// TIA Portal V17 export
// export: Created 2025-01-08T13:55:36.0615865Z, ExportSetting WithDefaults, DisplayName Totally Integrated Automation Portal, DisplayVersion V17, DisplayName TIA Portal Openness, DisplayVersion V17, DisplayName TIA Portal Version Control Interface, DisplayVersion V17, DisplayName SINAMICS Startdrive Advanced, DisplayVersion V17 Update2, DisplayName SINAMICS Startdrive G130, G150, S120, S150, SINAMICS MV, S210, DisplayVersion V17 Update2, DisplayName SINAMICS Startdrive G110M, G120, G120C, G120D, G120P, G115D, DisplayVersion V17 Update2, DisplayName STEP 7 Professional, DisplayVersion V17, DisplayName STEP 7 Safety, DisplayVersion V17, DisplayName WinCC Advanced, DisplayVersion V17
TYPE "UDT_Subsystem_Utility"
// stored: IsFailsafeCompliant false
   STRUCT
      Lifebit : Bool;   // Lifebit 1Hz, Check data exchange
      Fault : Bool;   // General Fault
      active : Bool;   // Machine is running or ready
      in_progress : Bool;   // Operation in is progress, motors are running
      EStop : Bool;   // Emergency stop active (1=good)
      General05 : Bool;   // General Signal, Operation mode 05
      General06 : Bool;   // General Signal, Operation mode 06
      General07 : Bool;   // General Signal, Operation mode 07
      General08 : Bool;   // General Signal, Operation mode 08
      General09 : Bool;   // General Signal, Operation mode 09
      General10 : Bool;   // General Signal, Operation mode 10
      General11 : Bool;   // General Signal, Operation mode 11
      General12 : Bool;   // General Signal, Operation mode 12
      General13 : Bool;   // General Signal, Operation mode 13
      General14 : Bool;   // General Signal, Operation mode 14
      General15 : Bool;   // General Signal, Operation mode 15
      Status00 : Bool;   // Motor running, status 00
      Status01 : Bool;   // Motor running, status 01
      Status02 : Bool;   // Motor running, status 02
      Status03 : Bool;   // Motor running, status 03
      Status04 : Bool;   // Motor running, status 04
      Status05 : Bool;   // Motor running, status 05
      Status06 : Bool;   // Motor running, status 06
      Status07 : Bool;   // Motor running, status 07
      Status08 : Bool;   // Motor running, status 08
      Status09 : Bool;   // Motor running, status 09
      Status10 : Bool;   // Motor running, status 10
      Status11 : Bool;   // Motor running, status 11
      Status12 : Bool;   // Motor running, status 12
      Status13 : Bool;   // Motor running, status 13
      Status14 : Bool;   // Motor running, status 14
      Status15 : Bool;   // Motor running, status 15
      Status16 : Bool;   // Motor running, status 16
      Status17 : Bool;   // Motor running, status 17
      Status18 : Bool;   // Motor running, status 18
      Status19 : Bool;   // Motor running, status 19
      Status20 : Bool;   // Motor running, status 20
      Status21 : Bool;   // Motor running, status 21
      Status22 : Bool;   // Motor running, status 22
      Status23 : Bool;   // Motor running, status 23
      Status24 : Bool;   // Motor running, status 24
      Status25 : Bool;   // Motor running, status 25
      Status26 : Bool;   // Motor running, status 26
      Status27 : Bool;   // Motor running, status 27
      Status28 : Bool;   // Motor running, status 28
      Status29 : Bool;   // Motor running, status 29
      Status30 : Bool;   // Motor running, status 30
      Status31 : Bool;   // Motor running, status 31
      Alarm000 : Bool;   // Alarm 0 active
      Alarm001 : Bool;   // Alarm 1 active
      Alarm002 : Bool;   // Alarm 2 active
      Alarm003 : Bool;   // Alarm 3 active
      Alarm004 : Bool;   // Alarm 4 active
      Alarm005 : Bool;   // Alarm 5 active
      Alarm006 : Bool;   // Alarm 6 active
      Alarm007 : Bool;   // Alarm 7 active
      Alarm008 : Bool;   // Alarm 8 active
      Alarm009 : Bool;   // Alarm 9 active
      Alarm010 : Bool;   // Alarm 10 active
      Alarm011 : Bool;   // Alarm 11 active
      Alarm012 : Bool;   // Alarm 12 active
      Alarm013 : Bool;   // Alarm 13 active
      Alarm014 : Bool;   // Alarm 14 active
      Alarm015 : Bool;   // Alarm 15 active
      Alarm016 : Bool;   // Alarm 16 active
      Alarm017 : Bool;   // Alarm 17 active
      Alarm018 : Bool;   // Alarm 18 active
      Alarm019 : Bool;   // Alarm 19 active
      Alarm020 : Bool;   // Alarm 20 active
      Alarm021 : Bool;   // Alarm 21 active
      Alarm022 : Bool;   // Alarm 22 active
      Alarm023 : Bool;   // Alarm 23 active
      Alarm024 : Bool;   // Alarm 24 active
      Alarm025 : Bool;   // Alarm 25 active
      Alarm026 : Bool;   // Alarm 26 active
      Alarm027 : Bool;   // Alarm 27 active
      Alarm028 : Bool;   // Alarm 28 active
      Alarm029 : Bool;   // Alarm 29 active
      Alarm030 : Bool;   // Alarm 30 active
      Alarm031 : Bool;   // Alarm 31 active
      Alarm032 : Bool;   // Alarm 32 active
      Alarm033 : Bool;   // Alarm 33 active
      Alarm034 : Bool;   // Alarm 34 active
      Alarm035 : Bool;   // Alarm 35 active
      Alarm036 : Bool;   // Alarm 36 active
      Alarm037 : Bool;   // Alarm 37 active
      Alarm038 : Bool;   // Alarm 38 active
      Alarm039 : Bool;   // Alarm 39 active
      Alarm040 : Bool;   // Alarm 40 active
      Alarm041 : Bool;   // Alarm 41 active
      Alarm042 : Bool;   // Alarm 42 active
      Alarm043 : Bool;   // Alarm 43 active
      Alarm044 : Bool;   // Alarm 44 active
      Alarm045 : Bool;   // Alarm 45 active
      Alarm046 : Bool;   // Alarm 46 active
      Alarm047 : Bool;   // Alarm 47 active
      Alarm048 : Bool;   // Alarm 48 active
      Alarm049 : Bool;   // Alarm 49 active
      Alarm050 : Bool;   // Alarm 50 active
      Alarm051 : Bool;   // Alarm 51 active
      Alarm052 : Bool;   // Alarm 52 active
      Alarm053 : Bool;   // Alarm 53 active
      Alarm054 : Bool;   // Alarm 54 active
      Alarm055 : Bool;   // Alarm 55 active
      Alarm056 : Bool;   // Alarm 56 active
      Alarm057 : Bool;   // Alarm 57 active
      Alarm058 : Bool;   // Alarm 58 active
      Alarm059 : Bool;   // Alarm 59 active
      Alarm060 : Bool;   // Alarm 60 active
      Alarm061 : Bool;   // Alarm 61 active
      Alarm062 : Bool;   // Alarm 62 active
      Alarm063 : Bool;   // Alarm 63 active
      Alarm064 : Bool;   // Alarm 64 active
      Alarm065 : Bool;   // Alarm 65 active
      Alarm066 : Bool;   // Alarm 66 active
      Alarm067 : Bool;   // Alarm 67 active
      Alarm068 : Bool;   // Alarm 68 active
      Alarm069 : Bool;   // Alarm 69 active
      Alarm070 : Bool;   // Alarm 70 active
      Alarm071 : Bool;   // Alarm 71 active
      Alarm072 : Bool;   // Alarm 72 active
      Alarm073 : Bool;   // Alarm 73 active
      Alarm074 : Bool;   // Alarm 74 active
      Alarm075 : Bool;   // Alarm 75 active
      Alarm076 : Bool;   // Alarm 76 active
      Alarm077 : Bool;   // Alarm 77 active
      Alarm078 : Bool;   // Alarm 78 active
      Alarm079 : Bool;   // Alarm 79 active
      Alarm080 : Bool;   // Alarm 80 active
      Alarm081 : Bool;   // Alarm 81 active
      Alarm082 : Bool;   // Alarm 82 active
      Alarm083 : Bool;   // Alarm 83 active
      Alarm084 : Bool;   // Alarm 84 active
      Alarm085 : Bool;   // Alarm 85 active
      Alarm086 : Bool;   // Alarm 86 active
      Alarm087 : Bool;   // Alarm 87 active
      Alarm088 : Bool;   // Alarm 88 active
      Alarm089 : Bool;   // Alarm 89 active
      Alarm090 : Bool;   // Alarm 90 active
      Alarm091 : Bool;   // Alarm 91 active
      Alarm092 : Bool;   // Alarm 92 active
      Alarm093 : Bool;   // Alarm 93 active
      Alarm094 : Bool;   // Alarm 94 active
      Alarm095 : Bool;   // Alarm 95 active
      Alarm096 : Bool;   // Alarm 96 active
      Alarm097 : Bool;   // Alarm 97 active
      Alarm098 : Bool;   // Alarm 98 active
      Alarm099 : Bool;   // Alarm 99 active
      Alarm100 : Bool;   // Alarm 100 active
      Alarm101 : Bool;   // Alarm 101 active
      Alarm102 : Bool;   // Alarm 102 active
      Alarm103 : Bool;   // Alarm 103 active
      Alarm104 : Bool;   // Alarm 104 active
      Alarm105 : Bool;   // Alarm 105 active
      Alarm106 : Bool;   // Alarm 106 active
      Alarm107 : Bool;   // Alarm 107 active
      Alarm108 : Bool;   // Alarm 108 active
      Alarm109 : Bool;   // Alarm 109 active
      Alarm110 : Bool;   // Alarm 110 active
      Alarm111 : Bool;   // Alarm 111 active
      Alarm112 : Bool;   // Alarm 112 active
      Alarm113 : Bool;   // Alarm 113 active
      Alarm114 : Bool;   // Alarm 114 active
      Alarm115 : Bool;   // Alarm 115 active
      Alarm116 : Bool;   // Alarm 116 active
      Alarm117 : Bool;   // Alarm 117 active
      Alarm118 : Bool;   // Alarm 118 active
      Alarm119 : Bool;   // Alarm 119 active
      Alarm120 : Bool;   // Alarm 120 active
      Alarm121 : Bool;   // Alarm 121 active
      Alarm122 : Bool;   // Alarm 122 active
      Alarm123 : Bool;   // Alarm 123 active
      Alarm124 : Bool;   // Alarm 124 active
      Alarm125 : Bool;   // Alarm 125 active
      Alarm126 : Bool;   // Alarm 126 active
      Alarm127 : Bool;   // Alarm 127 active
      OperatingHours : DWord;   // Operating hours of machine
      DownTimeHours : DWord;   // Downtime hours of machine
      Speed : Word;   // Production speed
      Container_total : DWord;   // Container counter of the actual batch.
      Container_good : DWord;   // Good container counter
      Container_reject : DWord;   // rejected container counter
      Counter_06 : DWord;   // Counter 06
      Counter_07 : DWord;   // Counter 07
      Counter_08 : DWord;   // Counter 08
      Counter_09 : DWord;   // Counter 09
      Counter_10 : DWord;   // Counter 10
      Counter_11 : DWord;   // Counter 11
      Total_Amount : Real;   // Total filling amount of the actual batch. [kg]
      Amount_01 : Real;   // Amount 01
      Amount_02 : Real;   // Amount 02
      Amount_03 : Real;   // Amount 03
      FormatName : String[20];
   END_STRUCT;
END_TYPE
